(* PLC project SafeLOGIC-1, BrAutomation SafeDESIGNER  4.3.4.4 *)
(* stored: companyURL http://www.br-automation.com, creationDateTime Thu Jun 24 15:47:40 2021 *)

PROGRAM Main
  VAR  (* added by the conversion: wires and edge detectors of the diagram *)
    _SAFEBOOL_TO_BOOL25_OUT : BOOL;
  END_VAR

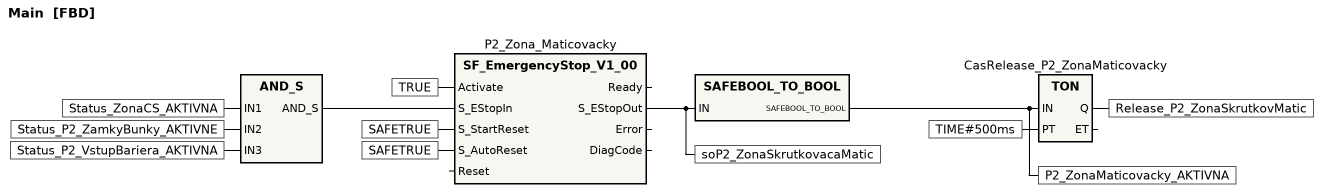
(* FBD diagram, written out as Structured Text *)
P2_Zona_Maticovacky(Activate := TRUE, S_EStopIn := AND_S(Status_ZonaCS_AKTIVNA, Status_P2_ZamkyBunky_AKTIVNE, Status_P2_VstupBariera_AKTIVNA), S_StartReset := SAFETRUE, S_AutoReset := SAFETRUE);
soP2_ZonaSkrutkovacaMatic := P2_Zona_Maticovacky.S_EStopOut;
_SAFEBOOL_TO_BOOL25_OUT := SAFEBOOL_TO_BOOL(P2_Zona_Maticovacky.S_EStopOut);
P2_ZonaMaticovacky_AKTIVNA := _SAFEBOOL_TO_BOOL25_OUT;
CasRelease_P2_ZonaMaticovacky(IN := _SAFEBOOL_TO_BOOL25_OUT, PT := TIME#500ms);
Release_P2_ZonaSkrutkovMatic := CasRelease_P2_ZonaMaticovacky.Q;
END_PROGRAM
